// TIA Portal V19 export
TYPE "LEXCHANGETRAY_typeVfd_monitor"
// stored: Access Published
   STRUCT
      vfd : "LBC_typeSinaSpeedControlNodeMonitoring";
      downloadStatus { S7_SetPoint := 'True'} : Int;   // Parameter Download Status (0:Idle, 1:In Progress, 2:Complete, -1:Error)
      statVfdSportsInc { S7_SetPoint := 'True'} : Int;   // VFD Sports Mode Increment Status
      simulated { S7_SetPoint := 'True'} : Bool;   // VFD Simulation Mode Status
   END_STRUCT;
END_TYPE
